TYPE UDT_BoxList :
STRUCT
	Box: ARRAY[0..64] OF UDT_BOX;
END_STRUCT
END_TYPE

(* stored: Version 1.1.0.1, ProductVersion 3.1.4022.16
   DUT UDT_BoxList: Id {7c663cfd-1b33-45e0-8b79-192a7cfac469} *)
